ADAPTER ADP_INDICATION (* Adapter Interface *)
  (* Standard: 61499-1 *)
  (* Version 0.0, 1/1/2023, Dmitrii, Flexbridge AB *)
  PACKAGE UAO.Hackathon;
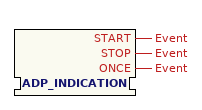
  EVENT_OUTPUT
    START; (* Request from Socket *)
    STOP; (* Response from Socket *)
    ONCE;
  END_EVENT
  SERVICE SOCKET/PLUG
    SEQUENCE request_confirm
      SOCKET.START(REQD) -> PLUG.START(REQD);
      PLUG.CNF(CNFD) -> SOCKET.CNF(CNFD);
    END_SEQUENCE
    SEQUENCE indication_response
      PLUG.IND(INDD) -> SOCKET.IND(INDD);
      SOCKET.STOP(RSPD) -> PLUG.STOP(RSPD);
    END_SEQUENCE
  END_SERVICE
END_ADAPTER
